FUNCTION_BLOCK CAT1 (* Composite Function Block Type *)
  (* Standard: 61499-2 *)
  (* Version 0.0, 2/19/2024, SESA658662, Schneider Electric, template *)
  PACKAGE Main;
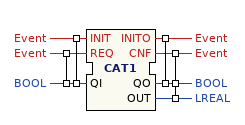
  EVENT_INPUT
    INIT WITH QI; (* Initialization Request *)
    REQ WITH QI; (* Normal Execution Request *)
  END_EVENT
  EVENT_OUTPUT
    INITO WITH QO; (* Initialization Confirm *)
    CNF WITH QO, OUT; (* Execution Confirmation *)
  END_EVENT
  VAR_INPUT
    QI : BOOL; (* Input event qualifier *)
  END_VAR
  VAR_OUTPUT
    QO : BOOL; (* Output event qualifier *)
    OUT : LREAL; (* Result: IN1 + IN2 + ... *)
  END_VAR
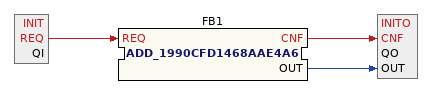
  FBS
    FB1 : ADD_1990CFD1468AAE4A6; {SET_ATTRIBUTE(Configuration.GenericFBType.InterfaceParams, Runtime.Standard#CNT:=2;IN${CNT$}:LREAL)}
  END_FBS
  EVENT_CONNECTIONS
    REQ TO FB1.REQ;
    FB1.CNF TO CNF;
  END_CONNECTIONS
  DATA_CONNECTIONS
    FB1.OUT TO OUT;
  END_CONNECTIONS
END_FUNCTION_BLOCK
